Staubli VAL3: getNum.pgx

public program getNum(string x_sTitle, num& x_nValue, num x_nMin, num x_nMax)
  local string l_sItemName
  local num l_nKey
  local num l_i
  local num l_nPos
  local num l_nValue
begin
  //获取一个数值
  l_nValue=x_nValue
  do
    call listframe(x_sTitle,10,5,20,1)
    call clear(11,6)
    gotoxy(15,6)
    l_nKey=get(l_nValue)
    //超出范围
    if l_nValue<x_nMin or l_nValue>x_nMax
      popUpMsg("取值范围:"+"["+toString(".3",x_nMin)+","+toString(".3",x_nMax)+"]")
      l_nValue=x_nValue
    else
      x_nValue=l_nValue
    endIf
    delay(0)
  until l_nKey==255

end
